TYPE ST_FeedPara :
STRUCT
	Width:UINT;
	Length:UINT;
	Thickness:REAL;
	Quantity :UINT;
	Groups:UINT;
	Total:UINT;
	
	FeedPOS1:REAL;
	FeedPOS2:REAL;
	
END_STRUCT
END_TYPE

(* stored: Version 1.1.0.1, ProductVersion 3.1.4024.15
   DUT ST_FeedPara: Id {015e7c2e-1f7d-46c3-972c-e4169c3b5a92} *)
